FUNCTION_BLOCK ThreeConCtlMulticast (* Composite Function Block Type *)
  (* Standard: 61499-2 *)
  (* Version 0.2, 2003-12-05, JHC, Rockwell Automation, Renamed from NEWCOMPFB. *)
  (* Version 0.1, 2002-01-08, JHC, Rockwell Automation, Added DLY FB as example. *)
  (* Version 0.0, 2000-05-27, JHC, Rockwell Automation *)
  (* Compiler header: package fb.rt.cs725; *)
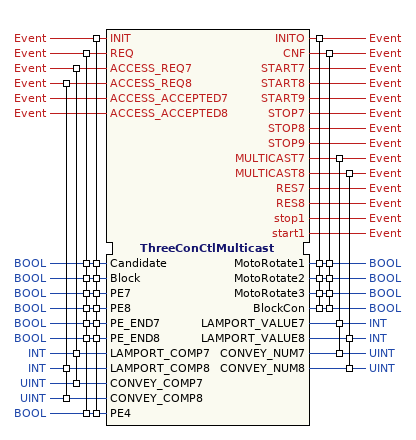
  EVENT_INPUT
    INIT WITH Candidate, Block, PE7, PE8, PE_END8, PE_END7, PE4; (* Initialization Request *)
    REQ WITH Block, Candidate, PE7, PE8, PE_END7, PE_END8, PE4; (* Normal Execution Request *)
    ACCESS_REQ7 WITH LAMPORT_COMP7, CONVEY_COMP7;
    ACCESS_REQ8 WITH LAMPORT_COMP8, CONVEY_COMP8;
    ACCESS_ACCEPTED7;
    ACCESS_ACCEPTED8;
  END_EVENT
  EVENT_OUTPUT
    INITO WITH MotoRotate1, MotoRotate2, MotoRotate3, BlockCon; (* Initialization Confirm *)
    CNF WITH MotoRotate1, MotoRotate2, MotoRotate3, BlockCon; (* Execution Confirmation *)
    START7;
    START8;
    START9;
    STOP7;
    STOP8;
    STOP9;
    MULTICAST7 WITH LAMPORT_VALUE7, CONVEY_NUM7;
    MULTICAST8 WITH CONVEY_NUM8, LAMPORT_VALUE8;
    RES7;
    RES8;
    stop1;
    start1;
  END_EVENT
  VAR_INPUT
    Candidate : BOOL;
    Block : BOOL;
    PE7 : BOOL;
    PE8 : BOOL;
    PE_END7 : BOOL;
    PE_END8 : BOOL;
    LAMPORT_COMP7 : INT;
    LAMPORT_COMP8 : INT;
    CONVEY_COMP7 : UINT;
    CONVEY_COMP8 : UINT;
    PE4 : BOOL;
  END_VAR
  VAR_OUTPUT
    MotoRotate1 : BOOL;
    MotoRotate2 : BOOL;
    MotoRotate3 : BOOL;
    BlockCon : BOOL;
    LAMPORT_VALUE7 : INT;
    LAMPORT_VALUE8 : INT;
    CONVEY_NUM7 : UINT;
    CONVEY_NUM8 : UINT;
  END_VAR
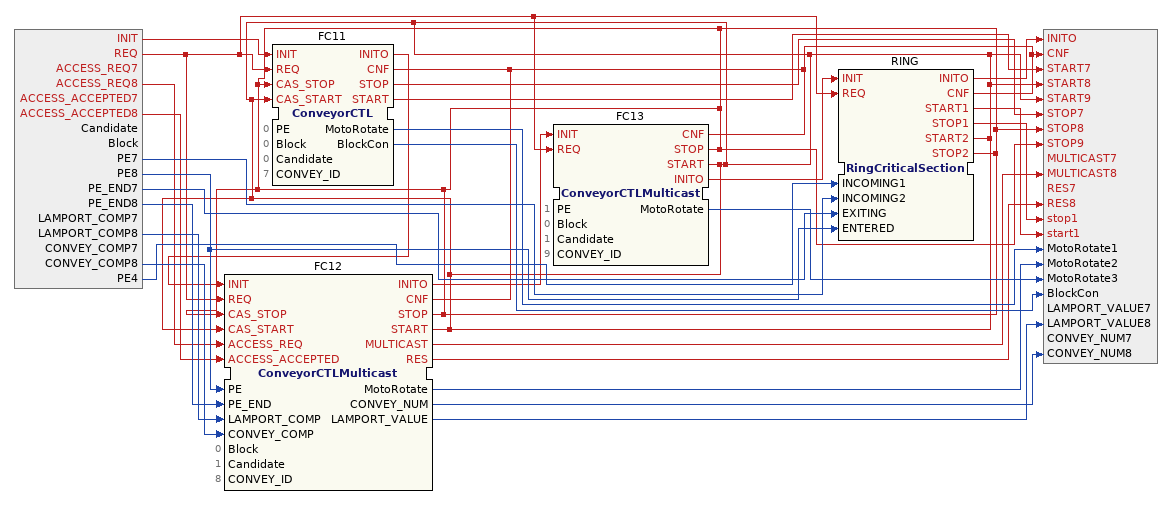
  FBS
    FC11 : ConveyorCTL(CONVEY_ID := 7, PE := 0, Block := 0, Candidate := 0);
    FC12 : ConveyorCTLMulticast(Block := 0, Candidate := 1, CONVEY_ID := 8);
    FC13 : ConveyorCTLMulticast(PE := 1, Block := 0, Candidate := 1, CONVEY_ID := 9);
    RING : RingCriticalSection;
  END_FBS
  EVENT_CONNECTIONS
    INIT TO FC11.INIT;
    REQ TO FC11.REQ;
    FC11.INITO TO FC12.INIT;
    FC12.INITO TO FC13.INIT;
    FC13.CNF TO CNF;
    REQ TO FC12.REQ;
    REQ TO FC13.REQ;
    FC11.CNF TO CNF;
    FC12.CNF TO CNF;
    FC12.STOP TO STOP8;
    FC11.STOP TO STOP7;
    FC13.STOP TO STOP9;
    FC13.STOP TO FC11.CAS_STOP;
    FC13.STOP TO FC12.CAS_STOP;
    FC12.STOP TO FC11.CAS_STOP;
    FC13.START TO START9;
    FC11.START TO START7;
    FC12.START TO START8;
    FC12.START TO FC11.CAS_START;
    FC13.START TO FC11.CAS_START;
    FC13.START TO FC12.CAS_START;
    FC12.MULTICAST TO MULTICAST8;
    FC12.RES TO RES8;
    ACCESS_REQ8 TO FC12.ACCESS_REQ;
    ACCESS_ACCEPTED8 TO FC12.ACCESS_ACCEPTED;
    RING.INITO TO INITO;
    FC13.INITO TO RING.INIT;
    REQ TO RING.REQ;
    RING.CNF TO CNF;
    RING.START1 TO start1;
    RING.STOP1 TO stop1;
    RING.START2 TO FC11.CAS_START;
    RING.STOP2 TO FC11.CAS_STOP;
  END_CONNECTIONS
  DATA_CONNECTIONS
    FC13.MotoRotate TO MotoRotate3;
    FC12.MotoRotate TO MotoRotate2;
    FC11.MotoRotate TO MotoRotate1;
    FC11.BlockCon TO BlockCon;
    PE8 TO FC12.PE;
    PE_END8 TO FC12.PE_END;
    LAMPORT_COMP8 TO FC12.LAMPORT_COMP;
    CONVEY_COMP8 TO FC12.CONVEY_COMP;
    FC12.CONVEY_NUM TO CONVEY_NUM8;
    FC12.LAMPORT_VALUE TO LAMPORT_VALUE8;
    PE7 TO RING.INCOMING2;
    PE4 TO RING.INCOMING1;
    PE_END7 TO RING.EXITING;
    PE8 TO RING.ENTERED;
  END_CONNECTIONS
END_FUNCTION_BLOCK
